{attribute 'qualified_only'}
{attribute 'strict'}
{attribute 'to_string'}
TYPE eGridMode :
(
	auto := 0,
	following := 1,
	forming	:= 2
);
END_TYPE

(* stored: Version 1.1.0.1, ProductVersion 3.1.4026.18
   DUT eGridMode: Id {461cb775-5766-4e6b-8f1d-75f8ea6aa313} *)
